FUNCTION_BLOCK PUBLIC FB_Foo
VAR_INPUT
END_VAR
VAR_OUTPUT
END_VAR
VAR
END_VAR

END_FUNCTION_BLOCK

(* stored: Version 1.1.0.1, ProductVersion 3.1.4020.6
   POU FB_Foo: Id {f7735ed4-7188-4d1c-99c9-3678af16f02d}, SpecialFunc None *)
